// TIA Portal V20 export
TYPE "LKinCtrl_typeCircleParameters"
   STRUCT
      circMode : DInt := 0;   // 0: auxPoint defines point on circle line; 1: auxPoint defines circle center; 2: radius and endPoint define circle segment; 3: GCode notation (end & aux point)
      point : DInt := -1;   // reference to point table, used for auxPoint
      auxPoint : Array[1..3] of LReal;   // auxiliary point for circle definition
      pathChoice : DInt := 0;   // circMode(0): not relevant; circMode(1): 0: pos direction; 1: neg direction; circMode(2): 0: short pos segment; 1: short neg segment; 2: long pos segment; 3: long neg segment
      circlePlane : DInt;   // circMode(0): not relevant; circMode(1+2): 0: XZ; 1: YZ; 2: XY
      radius : LReal;   // only in combination with circMode(2): radius
      arc : LReal;   // only in combination with circMode(1): arc
   END_STRUCT;
END_TYPE
